{attribute 'qualified_only'}
TYPE E_CylinderCommand : (NONE := 0, EXTEND := 1, RETRACT := 2) DINT;
END_TYPE

(* stored: Version 1.1.0.1, ProductVersion 3.1.4024.12
   DUT E_CylinderCommand: Id {73e68c86-09bd-4865-9c57-a7e1156f5c00} *)
